PROGRAM MAIN
VAR
	rawValue		:REAL := 100;		// This can be a sensor
	
	rFilterSize		:REAL := 0.99;
	rFilteredValue	:REAL;
	bError 			:BOOL;
END_VAR

bError := fnSimpleFilter(UnfilterdValue := rawValue, FilterSize := rFilterSize, FilteredValue := rFilteredValue);

END_PROGRAM

(* stored: Version 1.1.0.1, ProductVersion 3.1.4024.13
   POU MAIN: Id {80972c77-6d86-4e71-8266-5973a4116248}, SpecialFunc None *)
